{attribute 'linkalways'} 
{attribute 'no_explicit_call' := 'This FB is a CLASS and must be accessed using methods or properties'}
{attribute 'enable_dynamic_creation'}
FUNCTION_BLOCK Node_F_VN_GetImageChannel EXTENDS VisionNode
VAR
    ipSrcImage : _ITcVnImage;
    ipDestImage : _ITcVnImage;
    nChannelIndex : _UINT(0);
    hrPrev : _HRESULT(S_OK);
	hresult : _HRESULT(S_OK);
END_VAR

METHOD PUBLIC  Clone : I_Node
VAR
	pNode : POINTER TO Node_F_VN_GetImageChannel;
END_VAR
pNode := __NEW(Node_F_VN_GetImageChannel);
Clone := pNode^;
END_METHOD

METHOD FB_init : BOOL
VAR_INPUT
	bInitRetains : BOOL; // if TRUE, the retain variables are initialized (warm start / cold start)
	bInCopyCode : BOOL;  // if TRUE, the instance afterwards gets moved into the copy code (online change)
END_VAR
AddInput('ipSrcImage', ipSrcImage);
AddInput('hrPrev', hrPrev);
AddOutput('ipDestImage', ipDestImage);
AddOutput('hresult',hresult);
AddParameter('nChannelIndex', nChannelIndex);
END_METHOD

METHOD PROTECTED OnExecute
// ----------------------------------------------------------------------------
// TcVision 4.0.6.5 BUG FIX
// ----------------------------------------------------------------------------
// Get Image Channel fails, if used on two different sized images, 
// without clearing the destination image first. 
// so, we check to see if hrPrev is failed, in which case we do nothing
// as the function would do nothing natively.  Else, we check the dest
// image, and if it has something, it is first emptied
// ---------------------------------------------------------------------------- 
IF failed(hrPrev.Value) THEN
	RETURN;
END_IF

IF ipDestImage.IsValid THEN
	ipDestImage.Value.TcRelease();
	ipDestImage.Value := 0;
END_IF
// ---------------------------------------------------------------------------- 

hresult.Value := F_VN_GetImageChannel(
    ipSrcImage := ipSrcImage.Value,
	ipDestImage := ipDestImage.Value,
    nChannelIndex := nChannelIndex.Value,
	hrPrev:= hrPrev.Value);
END_METHOD

METHOD PUBLIC PreExecutionCheck
VAR_INPUT
	Check : I_PreExecutionChecks;
END_VAR
Check.IsTrue(ipSrcImage.IsValid, 'ipSrcImage must contain an image');
END_METHOD

END_FUNCTION_BLOCK

(* stored: Version 1.1.0.1, ProductVersion 3.1.4024.15
   POU Node_F_VN_GetImageChannel: Id {e3fb07bb-f62e-08aa-14bb-bf4a14957dea}, SpecialFunc None
   Folder Constructor: Id {7cd41bff-6d37-006f-1b71-84ddb7ed915a}
   Method Clone: Id {9baffbd9-52de-04ed-382e-312661fb1f98}
   Method FB_init: Id {bad1c400-fed7-0819-3625-710b215f8024}
   Method OnExecute: Id {b37a9723-2623-069a-1441-85c9d871bc73}
   Method PreExecutionCheck: Id {e3d19fed-40ed-03e7-0843-6a223f32938b} *)
